(*
SPDX-FileCopyrightText: Â© 2026 Oleksandr Tiutyk <trofimich@gmail.com>
SPDX-License-Identifier: MIT
License: https://opensource.org/license/mit
*)

(*!
<summary>Defines global configuration parameters for the automation framework.</summary>
*)

{attribute 'qualified_only'}
VAR_GLOBAL CONSTANT
	(*! <summary>Default timeout duration for component initialization phase (5 seconds).</summary> *)
	InitializationTimeout : TIME := T#5S;
END_VAR

(* stored: Version 1.1.0.1
   GVL Parameters: Id {cd7a6ad5-ab90-4d05-92c3-8e49481d33c0}, ParameterList True *)
